{attribute 'GeneratedUsingTerminal: ELM2642-0000-0016'}
{attribute addProperty BoxType "ELM2642-0000-0016"}
{attribute addProperty Id "Outputs_Channel_2AT %Q*Outputs_Channel_78994C084"}
{attribute addProperty CRC "808709989"}
{attribute addProperty Size "4"}
TYPE DO_Group_2_Outputs_3033EF65 EXTENDS OutputBase_10CEE7DE :
STRUCT
	{attribute addProperty Name "Outputs_Channel_2"}
	Outputs_Channel_2 AT %Q* : Outputs_Channel_78994C08;
END_STRUCT
END_TYPE

(* stored: Version 1.2.0.0, ProductVersion 3.1.4024.9
   DUT DO_Group_2_Outputs_3033EF65: Id {3cffe8bf-bae3-44ac-9b6d-f5d479beedb5} *)
